INTERFACE I_DOGroup

// Add output to group
METHOD AddOutput
VAR_INPUT
	IDO			: I_DigitalOut;		// Digital output
END_VAR
END_METHOD

// Gets the total number of IOs in the group
PROPERTY Count : INT
GET
END_GET
END_PROPERTY

// Get a specific output from the group
METHOD GetOutput : I_DigitalOut
VAR_INPUT
	nOutputIndex		: INT;		// Output index
END_VAR
END_METHOD

// Set the command to the outputs in the group
METHOD SetCommand
VAR_INPUT
	eCommand	: E_DOCommand;
END_VAR
END_METHOD

END_INTERFACE

(* stored: Version 1.1.0.1, ProductVersion 3.1.4024.11
   Itf I_DOGroup: Id {77cdbb6a-b25c-44fd-9c61-0e16924037f0}
   Folder Methods: Id {c84e9588-7a66-4a33-9241-552f324e39ed}
   Folder Properties: Id {8aa7c5a5-3349-45b5-af16-bc18d0b7554d}
   Method AddOutput: Id {e4f61fde-6f06-4388-aa68-e03a1c9bc0da}
   Property Count: Id {16ac6071-69f8-45bd-b746-e20198552638}
   Get Get: Id {46ce07e3-042d-4a61-ba1b-6fb7022e056b}
   Method GetOutput: Id {dfa660dd-3bdb-4bb4-8dda-b1f06f4ac57d}
   Method SetCommand: Id {02fefac4-05e6-451c-988c-af2639752daa} *)
